FUNCTION F_DT_ToString : STRING
VAR_INPUT
	in:DATE_AND_TIME;
END_VAR
VAR
	tsDtToConvert:TIMESTRUCT;
END_VAR

tsDtToConvert:= DT_TO_SYSTEMTIME(in);

F_DT_ToString:= CONCAT(WORD_TO_STRING(tsDtToConvert.wDay),'/');
F_DT_ToString:= CONCAT(F_DT_ToString, CONCAT( WORD_TO_STRING(tsDtToConvert.wMonth),'/'));
F_DT_ToString:= CONCAT(F_DT_ToString, CONCAT( WORD_TO_STRING(tsDtToConvert.wYear),'/'));
F_DT_ToString:= CONCAT(F_DT_ToString, ' ');
F_DT_ToString:= CONCAT(F_DT_ToString, CONCAT( WORD_TO_STRING(tsDtToConvert.wHour),':'));
F_DT_ToString:= CONCAT(F_DT_ToString, CONCAT( WORD_TO_STRING(tsDtToConvert.wMinute),':'));
F_DT_ToString:= CONCAT(F_DT_ToString,  WORD_TO_STRING(tsDtToConvert.wSecond));

END_FUNCTION

(* stored: Version 1.1.0.1, ProductVersion 3.1.4020.12
   POU F_DT_ToString: Id {927214c1-1be2-4b2e-8062-ad6190bfce41}, SpecialFunc None *)
